FUNCTION F_Zbm1 : Real
VAR_INPUT
END_VAR
VAR
	Hm1: LREAL;
END_VAR
VAR CONSTANT
	bZm1 : REAL:=733.772//m
END_VAR

//Hm1 = 1400000+mr1k1 ben Y up
F_Hm1:= 1400000+M12.fPosition;

END_FUNCTION

(* stored: Version 1.1.0.1, ProductVersion 3.1.4022.12
   POU F_Zbm1: Id {71033c13-fe06-4a4a-b389-be39c96f346c}, SpecialFunc None *)
